PROGRAM P_MediaTransport
VAR
END_VAR

P_TableVacuum();
P_UpDownSlot();

END_PROGRAM

(* stored: Version 1.1.0.1, ProductVersion 3.1.4024.11
   POU P_MediaTransport: Id {ad0cf7d2-b7a2-42a0-ae27-07d98017670b}, SpecialFunc None *)
